// TIA Portal V19 export
DATA_BLOCK "Com_FromFruitPlantAlsafe"   // DB306
{ S7_Optimized_Access := 'TRUE' }
// stored: AutoNumber false, MemoryReserve 0
   VAR RETAIN
      AFM1 : Struct   // Signals To Ampack
         Prod_Fruit : Bool;   // Product available to supply Ampack
         Stop_Fruit : Bool;   // Information - Alsafe empty
         Bool_0_2 : Bool;
         Bool_0_3 : Bool;
         Bool_0_4 : Bool;
         Bool_0_5 : Bool;
         Bool_0_6 : Bool;
         Bool_0_7 : Bool;
         Sterile_Fruit : Bool;   // Alsafe and line to Ampack is in Sterile status
         RequestFlippingValveF1 : Bool;   // Request flipping lower seat valve cluster Filler 1
         Bool_1_2 : Bool;
         Bool_1_3 : Bool;
         Cleaning_Fruit : Bool;   // Alsafe and line to Ampack cleaning
         LineClean : Bool;   // Alsafe and line to Polygon clean
         Bool_1_6 : Bool;
         Bool_1_7 : Bool;
         Bool_2_0 : Bool;
         Req_SteamBarrier_PD_Cl2 : Bool;   // Request steam barier during Alsafe ster pre doser cluster 2 - Fruit
         Bool_2_2 : Bool;
         Bool_2_3 : Bool;
         Bool_2_4 : Bool;
         Bool_2_5 : Bool;
         Bool_2_6 : Bool;
         Bool_2_7 : Bool;
         Bool_3_0 : Bool;
         Bool_3_1 : Bool;
         Bool_3_2 : Bool;
         Bool_3_3 : Bool;
         Bool_3_4 : Bool;
         Bool_3_5 : Bool;
         Bool_3_6 : Bool;
         Bool_3_7 : Bool;
         Bool_4_0 : Bool;
         Bool_4_1 : Bool;
         Bool_4_2 : Bool;
         Bool_4_3 : Bool;
         Bool_4_4 : Bool;
         Bool_4_5 : Bool;
         Bool_4_6 : Bool;
         Bool_4_7 : Bool;
         INT_6 : Int;
         INT_8 : Int;
         INT_10 : Int;
         INT_12 : Int;
         INT_14 : Int;
         INT_16 : Int;
         LOC_WD_CNT : Int;
      END_STRUCT;
      Spacer : Array[0..38] of Byte;
      DB_VAR : Int;   // Temporary placeholder variable
   END_VAR
BEGIN
END_DATA_BLOCK
